// TIA Portal V19 export
TYPE "C402_STU_SBO_TYPIC"
   STRUCT
      CMD { ExternalAccessible := 'False'; ExternalVisible := 'False'; ExternalWritable := 'False'} : USInt;   // Sturing positionering afsluitboom
      SNEL { ExternalAccessible := 'False'; ExternalVisible := 'False'; ExternalWritable := 'False'} : USInt;   // Sturing versneld
      VGV_TOE { ExternalAccessible := 'False'; ExternalVisible := 'False'; ExternalWritable := 'False'} : USInt;   // Vrijgave sluiten (verkeerslichten voldoende lang op Rood)
      VGV_VWA_TOE { ExternalAccessible := 'False'; ExternalVisible := 'False'; ExternalWritable := 'False'} : USInt;   // Vrijgave voorwaardelijk sluiten
   END_STRUCT;
END_TYPE
